TEXTLIST TextList_FootPedalstate
  0 = 'ready'
  100 = 'error'
   = ''
END_TEXTLIST

(* stored: Version 1.1.0.1, ProductVersion 3.1.4024.11
   TextList TextList_FootPedalstate: Id {c3dd695a-cdf4-4245-b5ce-6092a61c8ec1} *)
